# EPICS autosave request: iocs/vacuum/req/vacuum_settings.req
# Operator settings restored across IOC restarts
$(P):PMP1:RUN
$(P):VLV1:CMD
